TYPE MotorOutput :
STRUCT
	ConveyorForward : BOOL;
	ConveyorBackward : BOOL;
	ConveyorStop : BOOL;
	ConveyorSpeed : UDINT;
END_STRUCT
END_TYPE

(* stored: Version 1.1.0.1, ProductVersion 3.1.4024.9
   DUT MotorOutput: Id {b4f77477-6686-4417-b5bb-5708a574b7b0} *)
